(* CoDeSys 2.3 export: ST_ALARM.EXP *)

(* Data type *)
TYPE ST_ALARM :
STRUCT
	AlLen  : REAL;
	AlCnt  : WORD;
	TimeInit : STRING;
	TimeEnd  : STRING;

	Alarm  : BOOL;
	Adver  : BOOL;
	Text   : STRING;

	AlInit : BOOL;
	AlEnd  : BOOL;
END_STRUCT
END_TYPE
